{attribute addProperty BoxType "AT2050-0500-0018"}
{attribute addProperty Id "A_0095_AT2021_5250_0019_AT2021_5250AT2021_3DCFC8D064080"}
{attribute addProperty CRC "680868018"}
{attribute addProperty SizeInBites "640"}
{attribute addProperty SizeInBytes "80"}
TYPE A_0049_AT2050_0500_0018_289538B2 EXTENDS AT2050_9506A482 :
STRUCT
	{attribute addProperty Name "A_0095_AT2021_5250_0019_AT2021_5250"}
	A_0095_AT2021_5250_0019_AT2021_5250 : AT2021_3DCFC8D0;
END_STRUCT
END_TYPE

(* stored: Version 1.2.0.0, ProductVersion 3.1.4024.9
   DUT A_0049_AT2050_0500_0018_289538B2: Id {3bd119c8-2d2c-49e0-9674-d22a8df4d6d3} *)
